PROGRAM MAIN

Voyants();

_0_LASER_ST();
_1_LASER();
Defauts_Alarmes();
Parametres_PNC();
Status_machine();
Status_Ethercat();
 OK_Rep_Chariot_BE();
 OK_Rep_Pupitre();
 OK_Repartiteurs_Laser();
 Rep_BE();
 Rep_Bs();
Regulation_Centrale_Hydro();
En_service();
Divers_cycles();
G7_General();
Ech_Com_Pupitre();
Pupitre();
_0_LASER_ST();
_1_LASER();
_Divers_lifter_VB();
Divers_Decoupe();
G7_Cycle_Percages_Laser();
G7_Sel_Face();
G7_Master_Palpages();
G7_Palpage_Capacitance();
G7_Palpage_Sommet_L();
Presseurs_Laser();
Gestion_Pince();
Axe_01_X();
Axe_02_ZChariot();
Axe_03_X_Laser();
Axe_04_Y_Laser();
Axe_05_Z_Laser();
Axe_06_A();
Divers_axe();
Exec_ISO();

Forcage_Rep();
Gestion_ConvLaser();

END_PROGRAM

(* stored: Version 1.1.0.1
   POU MAIN: Id {b11d1c43-f64e-4f70-be59-2ceadac43aa4}, SpecialFunc None *)
